{attribute 'qualified_only'}
{attribute 'strict'}
TYPE E_Status :
(
	enum_member := 0
);
END_TYPE

(* stored: Version 1.1.0.1, ProductVersion 3.1.4024.10
   DUT E_Status: Id {94aa14c4-ba0f-46c4-9d24-09cbc08d6a64} *)
